{attribute 'linkalways'} 
{attribute 'no_explicit_call' := 'This FB is a CLASS and must be accessed using methods or properties'}
{attribute 'enable_dynamic_creation'}
FUNCTION_BLOCK FINAL RealDisplayNode EXTENDS Node
VAR
	in : _REAL(0.0);
	display : _REAL(0.0);
END_VAR

METHOD PUBLIC Clone : I_Node
VAR
	pNode : POINTER TO RealDisplayNode;
END_VAR
pNode := __NEW(RealDisplayNode);
Clone := pNode^;
END_METHOD

METHOD FB_init : BOOL
VAR_INPUT
	bInitRetains : BOOL; // if TRUE, the retain variables are initialized (warm start / cold start)
	bInCopyCode : BOOL;  // if TRUE, the instance afterwards gets moved into the copy code (online change)
END_VAR
AddInput('in', in);
AddContent('display', display);
END_METHOD

METHOD PROTECTED OnExecute : HRESULT
display.Value := in.Value;
END_METHOD

END_FUNCTION_BLOCK

(* stored: Version 1.1.0.1, ProductVersion 3.1.4024.12
   POU RealDisplayNode: Id {ee7f9bab-b57a-0c76-280a-ca9162805af7}, SpecialFunc None
   Folder Constructor: Id {cf4c5c7e-ac9a-09d3-1d02-93fbf4603598}
   Method Clone: Id {5e3d63f0-a052-00b2-22bc-bad220a790d3}
   Method FB_init: Id {eef82d27-df52-0ddf-104c-4ab2fd8161dc}
   Method OnExecute: Id {b22cd310-491b-07fa-2223-e61fa3ca416d} *)
